   1:  PR[91,1] = PR[90,1] + 0.629;
   1:L PR[91] R[100]mm/sec CNT100;
   1:  PR[91,1] = PR[90,1] + 1.561;
   1:  PR[91,2] = PR[90,2] + -23.325;
   1:L PR[91] R[100]mm/sec CNT100;
   1:  PR[91,1] = PR[90,1] + 7.477;
   1:  PR[91,2] = PR[90,2] + -23.910;
   1:L PR[91] R[100]mm/sec CNT100;
   1:  PR[91,1] = PR[90,1] + 8.164;
   1:  PR[91,2] = PR[90,2] + -23.821;
   1:L PR[91] R[100]mm/sec CNT100;
   1:  PR[91,1] = PR[90,1] + 13.666;
   1:  PR[91,2] = PR[90,2] + -22.946;
   1:L PR[91] R[100]mm/sec CNT100;
   1:  PR[91,1] = PR[90,1] + 14.550;
   1:  PR[91,2] = PR[90,2] + -22.590;
   1:L PR[91] R[100]mm/sec CNT100;
   1:  PR[91,1] = PR[90,1] + 19.392;
   1:  PR[91,2] = PR[90,2] + -20.484;
   1:L PR[91] R[100]mm/sec CNT100;
   1:  PR[91,1] = PR[90,1] + 20.346;
   1:  PR[91,2] = PR[90,2] + -19.776;
   1:L PR[91] R[100]mm/sec CNT100;
   1:  PR[91,1] = PR[90,1] + 24.273;
   1:  PR[91,2] = PR[90,2] + -16.705;
   1:L PR[91] R[100]mm/sec CNT100;
   1:  PR[91,1] = PR[90,1] + 25.132;
   1:  PR[91,2] = PR[90,2] + -15.619;
   1:L PR[91] R[100]mm/sec CNT100;
   1:  PR[91,1] = PR[90,1] + 28.000;
   1:  PR[91,2] = PR[90,2] + -11.846;
   1:L PR[91] R[100]mm/sec CNT100;
   1:  PR[91,1] = PR[90,1] + 28.598;
   1:  PR[91,2] = PR[90,2] + -10.471;
   1:L PR[91] R[100]mm/sec CNT100;
   1:  PR[91,1] = PR[90,1] + 30.330;
   1:  PR[91,2] = PR[90,2] + -6.297;
   1:L PR[91] R[100]mm/sec CNT100;
   1:  PR[91,1] = PR[90,1] + 30.542;
   1:  PR[91,2] = PR[90,2] + -4.725;
   1:L PR[91] R[100]mm/sec CNT100;
   1:  PR[91,1] = PR[90,1] + 30.756;
   1:  PR[91,2] = PR[90,2] + -2.568;
   1:L PR[91] R[100]mm/sec CNT100;
   1:  PR[91,1] = PR[90,1] + 31.056;
   1:  PR[91,2] = PR[90,2] + -0.286;
   1:L PR[91] R[100]mm/sec CNT100;
   1:  PR[91,1] = PR[90,1] + 30.904;
   1:  PR[91,2] = PR[90,2] + 1.310;
   1:L PR[91] R[100]mm/sec CNT100;
   1:  PR[91,1] = PR[90,1] + 30.330;
   1:  PR[91,2] = PR[90,2] + 5.670;
   1:L PR[91] R[100]mm/sec CNT100;
   1:  PR[91,1] = PR[90,1] + 28.603;
   1:  PR[91,2] = PR[90,2] + 9.838;
   1:L PR[91] R[100]mm/sec CNT100;
   1:  PR[91,1] = PR[90,1] + 28.006;
   1:  PR[91,2] = PR[90,2] + 11.211;
   1:L PR[91] R[100]mm/sec CNT100;
   1:  PR[91,1] = PR[90,1] + 25.143;
   1:  PR[91,2] = PR[90,2] + 14.983;
   1:L PR[91] R[100]mm/sec CNT100;
   1:  PR[91,1] = PR[90,1] + 24.286;
   1:  PR[91,2] = PR[90,2] + 16.068;
   1:L PR[91] R[100]mm/sec CNT100;
   1:  PR[91,1] = PR[90,1] + 20.366;
   1:  PR[91,2] = PR[90,2] + 19.139;
   1:L PR[91] R[100]mm/sec CNT100;
   1:  PR[91,1] = PR[90,1] + 19.413;
   1:  PR[91,2] = PR[90,2] + 19.847;
   1:L PR[91] R[100]mm/sec CNT100;
   1:  PR[91,1] = PR[90,1] + 14.579;
   1:  PR[91,2] = PR[90,2] + 21.956;
   1:L PR[91] R[100]mm/sec CNT100;
   1:  PR[91,1] = PR[90,1] + 13.695;
   1:  PR[91,2] = PR[90,2] + 22.313;
   1:L PR[91] R[100]mm/sec CNT100;
   1:  PR[91,1] = PR[90,1] + 8.201;
   1:  PR[91,2] = PR[90,2] + 23.194;
   1:L PR[91] R[100]mm/sec CNT100;
   1:  PR[91,1] = PR[90,1] + 7.513;
   1:  PR[91,2] = PR[90,2] + 23.285;
   1:L PR[91] R[100]mm/sec CNT100;
   1:  PR[91,1] = PR[90,1] + 1.597;
   1:  PR[91,2] = PR[90,2] + 22.714;
   1:L PR[91] R[100]mm/sec CNT100;
   1:  PR[91,1] = PR[90,1] + 1.222;
   1:  PR[91,2] = PR[90,2] + 22.667;
   1:L PR[91] R[100]mm/sec CNT100;
   1:  PR[91,1] = PR[90,1] + 0.703;
   1:  PR[91,2] = PR[90,2] + 22.501;
   1:L PR[91] R[100]mm/sec CNT100;
   1:  PR[91] = PR[90];
   1:  PR[91,1] = PR[90,1] + -0.529;
   1:  PR[91,2] = PR[90,2] + 22.670;
   1:  PR[91,3] = PR[90,3] + 57.035;
   1:L PR[91] R[100]mm/sec CNT100;
   1:  PR[91,1] = PR[90,1] + -0.847;
   1:  PR[91,2] = PR[90,2] + 22.772;
   1:L PR[91] R[100]mm/sec CNT100;
   1:  PR[91,1] = PR[90,1] + -0.976;
   1:  PR[91,2] = PR[90,2] + 22.788;
   1:L PR[91] R[100]mm/sec CNT100;
   1:  PR[91,1] = PR[90,1] + -7.156;
   1:  PR[91,2] = PR[90,2] + 23.384;
   1:L PR[91] R[100]mm/sec CNT100;
   1:  PR[91,1] = PR[90,1] + -7.594;
   1:  PR[91,2] = PR[90,2] + 23.327;
   1:L PR[91] R[100]mm/sec CNT100;
   1:  PR[91,1] = PR[90,1] + -13.353;
   1:  PR[91,2] = PR[90,2] + 22.404;
   1:L PR[91] R[100]mm/sec CNT100;
   1:  PR[91,1] = PR[90,1] + -13.996;
   1:  PR[91,2] = PR[90,2] + 22.143;
   1:L PR[91] R[100]mm/sec CNT100;
   1:  PR[91,1] = PR[90,1] + -19.083;
   1:  PR[91,2] = PR[90,2] + 19.924;
   1:L PR[91] R[100]mm/sec CNT100;
   1:  PR[91,1] = PR[90,1] + -19.826;
   1:  PR[91,2] = PR[90,2] + 19.372;
   1:L PR[91] R[100]mm/sec CNT100;
   1:  PR[91,1] = PR[90,1] + -23.967;
   1:  PR[91,2] = PR[90,2] + 16.128;
   1:L PR[91] R[100]mm/sec CNT100;
   1:  PR[91,1] = PR[90,1] + -24.660;
   1:  PR[91,2] = PR[90,2] + 15.252;
   1:L PR[91] R[100]mm/sec CNT100;
   1:  PR[91,1] = PR[90,1] + -27.694;
   1:  PR[91,2] = PR[90,2] + 11.258;
   1:L PR[91] R[100]mm/sec CNT100;
   1:  PR[91,1] = PR[90,1] + -28.187;
   1:  PR[91,2] = PR[90,2] + 10.118;
   1:L PR[91] R[100]mm/sec CNT100;
   1:  PR[91,1] = PR[90,1] + -30.024;
   1:  PR[91,2] = PR[90,2] + 5.680;
   1:L PR[91] R[100]mm/sec CNT100;
   1:  PR[91,1] = PR[90,1] + -30.201;
   1:  PR[91,2] = PR[90,2] + 4.374;
   1:L PR[91] R[100]mm/sec CNT100;
   1:  PR[91,1] = PR[90,1] + -30.383;
   1:  PR[91,2] = PR[90,2] + 2.537;
   1:L PR[91] R[100]mm/sec CNT100;
   1:  PR[91,1] = PR[90,1] + -30.761;
   1:  PR[91,2] = PR[90,2] + -0.338;
   1:L PR[91] R[100]mm/sec CNT100;
   1:  PR[91,1] = PR[90,1] + -30.632;
   1:  PR[91,2] = PR[90,2] + -1.679;
   1:L PR[91] R[100]mm/sec CNT100;
   1:  PR[91,1] = PR[90,1] + -30.021;
   1:  PR[91,2] = PR[90,2] + -6.312;
   1:L PR[91] R[100]mm/sec CNT100;
   1:  PR[91,1] = PR[90,1] + -28.182;
   1:  PR[91,2] = PR[90,2] + -10.752;
   1:L PR[91] R[100]mm/sec CNT100;
   1:  PR[91,1] = PR[90,1] + -27.688;
   1:  PR[91,2] = PR[90,2] + -11.893;
   1:L PR[91] R[100]mm/sec CNT100;
   1:  PR[91,1] = PR[90,1] + -24.649;
   1:  PR[91,2] = PR[90,2] + -15.889;
   1:L PR[91] R[100]mm/sec CNT100;
   1:  PR[91,1] = PR[90,1] + -23.954;
   1:  PR[91,2] = PR[90,2] + -16.765;
   1:L PR[91] R[100]mm/sec CNT100;
   1:  PR[91,1] = PR[90,1] + -19.805;
   1:  PR[91,2] = PR[90,2] + -20.009;
   1:L PR[91] R[100]mm/sec CNT100;
   1:  PR[91,1] = PR[90,1] + -19.062;
   1:  PR[91,2] = PR[90,2] + -20.560;
   1:L PR[91] R[100]mm/sec CNT100;
   1:  PR[91,1] = PR[90,1] + -13.967;
   1:  PR[91,2] = PR[90,2] + -22.777;
   1:L PR[91] R[100]mm/sec CNT100;
   1:  PR[91,1] = PR[90,1] + -13.323;
   1:  PR[91,2] = PR[90,2] + -23.036;
   1:L PR[91] R[100]mm/sec CNT100;
   1:  PR[91,1] = PR[90,1] + -7.557;
   1:  PR[91,2] = PR[90,2] + -23.953;
   1:L PR[91] R[100]mm/sec CNT100;
   1:  PR[91,1] = PR[90,1] + -7.120;
   1:  PR[91,2] = PR[90,2] + -24.009;
   1:L PR[91] R[100]mm/sec CNT100;
   1:  PR[91,1] = PR[90,1] + -0.879;
   1:  PR[91,2] = PR[90,2] + -23.392;
   1:L PR[91] R[100]mm/sec CNT100;
   1:  PR[91,1] = PR[90,1] + -0.799;
   1:  PR[91,2] = PR[90,2] + -23.382;
   1:L PR[91] R[100]mm/sec CNT100;
   1:  PR[91,1] = PR[90,1] + -0.525;
   1:  PR[91,2] = PR[90,2] + -23.296;
   1:L PR[91] R[100]mm/sec CNT100;
   1:  PR[91,1] = PR[90,1] + 0.614;
   1:L PR[91] R[100]mm/sec CNT100;
   1:  PR[91,1] = PR[90,1] + 1.097;
   1:  PR[91,2] = PR[90,2] + -23.398;
   1:L PR[91] R[100]mm/sec CNT100;
   1:  PR[91,1] = PR[90,1] + 7.278;
   1:  PR[91,2] = PR[90,2] + -24.009;
   1:L PR[91] R[100]mm/sec CNT100;
   1:  PR[91,1] = PR[90,1] + 7.716;
   1:  PR[91,2] = PR[90,2] + -23.953;
   1:L PR[91] R[100]mm/sec CNT100;
   1:  PR[91,1] = PR[90,1] + 13.481;
   1:  PR[91,2] = PR[90,2] + -23.036;
   1:L PR[91] R[100]mm/sec CNT100;
   1:  PR[91,1] = PR[90,1] + 14.126;
   1:  PR[91,2] = PR[90,2] + -22.776;
   1:L PR[91] R[100]mm/sec CNT100;
   1:  PR[91,1] = PR[90,1] + 19.220;
   1:  PR[91,2] = PR[90,2] + -20.561;
   1:L PR[91] R[100]mm/sec CNT100;
   1:  PR[91,1] = PR[90,1] + 19.963;
   1:  PR[91,2] = PR[90,2] + -20.009;
   1:L PR[91] R[100]mm/sec CNT100;
   1:  PR[91,1] = PR[90,1] + 24.111;
   1:  PR[91,2] = PR[90,2] + -16.765;
   1:L PR[91] R[100]mm/sec CNT100;
   1:  PR[91,1] = PR[90,1] + 24.806;
   1:  PR[91,2] = PR[90,2] + -15.887;
   1:L PR[91] R[100]mm/sec CNT100;
   1:  PR[91,1] = PR[90,1] + 27.845;
   1:  PR[91,2] = PR[90,2] + -11.889;
   1:L PR[91] R[100]mm/sec CNT100;
   1:  PR[91,1] = PR[90,1] + 28.340;
   1:  PR[91,2] = PR[90,2] + -10.752;
   1:L PR[91] R[100]mm/sec CNT100;
   1:  PR[91,1] = PR[90,1] + 30.179;
   1:  PR[91,2] = PR[90,2] + -6.318;
   1:L PR[91] R[100]mm/sec CNT100;
   1:  PR[91,1] = PR[90,1] + 30.357;
   1:  PR[91,2] = PR[90,2] + -5.007;
   1:L PR[91] R[100]mm/sec CNT100;
   1:  PR[91,1] = PR[90,1] + 30.539;
   1:  PR[91,2] = PR[90,2] + -3.166;
   1:L PR[91] R[100]mm/sec CNT100;
   1:  PR[91,1] = PR[90,1] + 30.918;
   1:  PR[91,2] = PR[90,2] + -0.286;
   1:L PR[91] R[100]mm/sec CNT100;
   1:  PR[91,1] = PR[90,1] + 30.790;
   1:  PR[91,2] = PR[90,2] + 1.057;
   1:L PR[91] R[100]mm/sec CNT100;
   1:  PR[91,1] = PR[90,1] + 30.180;
   1:  PR[91,2] = PR[90,2] + 5.690;
   1:L PR[91] R[100]mm/sec CNT100;
   1:  PR[91,1] = PR[90,1] + 28.344;
   1:  PR[91,2] = PR[90,2] + 10.118;
   1:L PR[91] R[100]mm/sec CNT100;
   1:  PR[91,1] = PR[90,1] + 27.851;
   1:  PR[91,2] = PR[90,2] + 11.254;
   1:L PR[91] R[100]mm/sec CNT100;
   1:  PR[91,1] = PR[90,1] + 24.817;
   1:  PR[91,2] = PR[90,2] + 15.251;
   1:L PR[91] R[100]mm/sec CNT100;
   1:  PR[91,1] = PR[90,1] + 24.123;
   1:  PR[91,2] = PR[90,2] + 16.128;
   1:L PR[91] R[100]mm/sec CNT100;
   1:  PR[91,1] = PR[90,1] + 19.983;
   1:  PR[91,2] = PR[90,2] + 19.372;
   1:L PR[91] R[100]mm/sec CNT100;
   1:  PR[91,1] = PR[90,1] + 19.241;
   1:  PR[91,2] = PR[90,2] + 19.924;
   1:L PR[91] R[100]mm/sec CNT100;
   1:  PR[91,1] = PR[90,1] + 14.154;
   1:  PR[91,2] = PR[90,2] + 22.143;
   1:L PR[91] R[100]mm/sec CNT100;
   1:  PR[91,1] = PR[90,1] + 13.511;
   1:  PR[91,2] = PR[90,2] + 22.403;
   1:L PR[91] R[100]mm/sec CNT100;
   1:  PR[91,1] = PR[90,1] + 7.752;
   1:  PR[91,2] = PR[90,2] + 23.327;
   1:L PR[91] R[100]mm/sec CNT100;
   1:  PR[91,1] = PR[90,1] + 7.314;
   1:  PR[91,2] = PR[90,2] + 23.384;
   1:L PR[91] R[100]mm/sec CNT100;
   1:  PR[91,1] = PR[90,1] + 1.135;
   1:  PR[91,2] = PR[90,2] + 22.788;
   1:L PR[91] R[100]mm/sec CNT100;
   1:  PR[91,1] = PR[90,1] + 1.006;
   1:  PR[91,2] = PR[90,2] + 22.772;
   1:L PR[91] R[100]mm/sec CNT100;
   1:  PR[91,1] = PR[90,1] + 0.688;
   1:  PR[91,2] = PR[90,2] + 22.670;
   1:L PR[91] R[100]mm/sec CNT100;
   1:  PR[91] = PR[90];
   1:  PR[91,1] = PR[90,1] + -0.359;
   1:  PR[91,2] = PR[90,2] + 22.840;
   1:  PR[91,3] = PR[90,3] + 57.645;
   1:L PR[91] R[100]mm/sec CNT100;
   1:  PR[91,1] = PR[90,1] + -6.957;
   1:  PR[91,2] = PR[90,2] + 23.484;
   1:L PR[91] R[100]mm/sec CNT100;
   1:  PR[91,1] = PR[90,1] + -7.145;
   1:  PR[91,2] = PR[90,2] + 23.459;
   1:L PR[91] R[100]mm/sec CNT100;
   1:  PR[91,1] = PR[90,1] + -13.168;
   1:  PR[91,2] = PR[90,2] + 22.494;
   1:L PR[91] R[100]mm/sec CNT100;
   1:  PR[91,1] = PR[90,1] + -13.572;
   1:  PR[91,2] = PR[90,2] + 22.330;
   1:L PR[91] R[100]mm/sec CNT100;
   1:  PR[91,1] = PR[90,1] + -18.911;
   1:  PR[91,2] = PR[90,2] + 20.001;
   1:L PR[91] R[100]mm/sec CNT100;
   1:  PR[91,1] = PR[90,1] + -19.443;
   1:  PR[91,2] = PR[90,2] + 19.605;
   1:L PR[91] R[100]mm/sec CNT100;
   1:  PR[91,1] = PR[90,1] + -23.805;
   1:  PR[91,2] = PR[90,2] + 16.189;
   1:L PR[91] R[100]mm/sec CNT100;
   1:  PR[91,1] = PR[90,1] + -24.335;
   1:  PR[91,2] = PR[90,2] + 15.519;
   1:L PR[91] R[100]mm/sec CNT100;
   1:  PR[91,1] = PR[90,1] + -27.539;
   1:  PR[91,2] = PR[90,2] + 11.301;
   1:L PR[91] R[100]mm/sec CNT100;
   1:  PR[91,1] = PR[90,1] + -27.929;
   1:  PR[91,2] = PR[90,2] + 10.399;
   1:L PR[91] R[100]mm/sec CNT100;
   1:  PR[91,1] = PR[90,1] + -29.874;
   1:  PR[91,2] = PR[90,2] + 5.701;
   1:L PR[91] R[100]mm/sec CNT100;
   1:  PR[91,1] = PR[90,1] + -30.015;
   1:  PR[91,2] = PR[90,2] + 4.655;
   1:L PR[91] R[100]mm/sec CNT100;
   1:  PR[91,1] = PR[90,1] + -30.166;
   1:  PR[91,2] = PR[90,2] + 3.133;
   1:L PR[91] R[100]mm/sec CNT100;
   1:  PR[91,1] = PR[90,1] + -30.622;
   1:  PR[91,2] = PR[90,2] + -0.338;
   1:L PR[91] R[100]mm/sec CNT100;
   1:  PR[91,1] = PR[90,1] + -30.518;
   1:  PR[91,2] = PR[90,2] + -1.427;
   1:L PR[91] R[100]mm/sec CNT100;
   1:  PR[91,1] = PR[90,1] + -29.871;
   1:  PR[91,2] = PR[90,2] + -6.333;
   1:L PR[91] R[100]mm/sec CNT100;
   1:  PR[91,1] = PR[90,1] + -27.923;
   1:  PR[91,2] = PR[90,2] + -11.033;
   1:L PR[91] R[100]mm/sec CNT100;
   1:  PR[91,1] = PR[90,1] + -27.533;
   1:  PR[91,2] = PR[90,2] + -11.936;
   1:L PR[91] R[100]mm/sec CNT100;
   1:  PR[91,1] = PR[90,1] + -24.323;
   1:  PR[91,2] = PR[90,2] + -16.156;
   1:L PR[91] R[100]mm/sec CNT100;
   1:  PR[91,1] = PR[90,1] + -23.792;
   1:  PR[91,2] = PR[90,2] + -16.826;
   1:L PR[91] R[100]mm/sec CNT100;
   1:  PR[91,1] = PR[90,1] + -19.423;
   1:  PR[91,2] = PR[90,2] + -20.242;
   1:L PR[91] R[100]mm/sec CNT100;
   1:  PR[91,1] = PR[90,1] + -18.890;
   1:  PR[91,2] = PR[90,2] + -20.637;
   1:L PR[91] R[100]mm/sec CNT100;
   1:  PR[91,1] = PR[90,1] + -13.543;
   1:  PR[91,2] = PR[90,2] + -22.964;
   1:L PR[91] R[100]mm/sec CNT100;
   1:  PR[91,1] = PR[90,1] + -13.139;
   1:  PR[91,2] = PR[90,2] + -23.126;
   1:L PR[91] R[100]mm/sec CNT100;
   1:  PR[91,1] = PR[90,1] + -7.108;
   1:  PR[91,2] = PR[90,2] + -24.085;
   1:L PR[91] R[100]mm/sec CNT100;
   1:  PR[91,1] = PR[90,1] + -6.921;
   1:  PR[91,2] = PR[90,2] + -24.109;
   1:L PR[91] R[100]mm/sec CNT100;
   1:  PR[91,1] = PR[90,1] + -0.762;
   1:  PR[91,2] = PR[90,2] + -23.500;
   1:L PR[91] R[100]mm/sec CNT100;
   1:  PR[91,1] = PR[90,1] + -0.352;
   1:  PR[91,2] = PR[90,2] + -23.464;
   1:L PR[91] R[100]mm/sec CNT100;
   1:  PR[91,1] = PR[90,1] + 0.519;
   1:L PR[91] R[100]mm/sec CNT100;
   1:  PR[91,1] = PR[90,1] + 7.079;
   1:  PR[91,2] = PR[90,2] + -24.109;
   1:L PR[91] R[100]mm/sec CNT100;
   1:  PR[91,1] = PR[90,1] + 7.266;
   1:  PR[91,2] = PR[90,2] + -24.085;
   1:L PR[91] R[100]mm/sec CNT100;
   1:  PR[91,1] = PR[90,1] + 13.297;
   1:  PR[91,2] = PR[90,2] + -23.125;
   1:L PR[91] R[100]mm/sec CNT100;
   1:  PR[91,1] = PR[90,1] + 13.701;
   1:  PR[91,2] = PR[90,2] + -22.963;
   1:L PR[91] R[100]mm/sec CNT100;
   1:  PR[91,1] = PR[90,1] + 19.048;
   1:  PR[91,2] = PR[90,2] + -20.638;
   1:L PR[91] R[100]mm/sec CNT100;
   1:  PR[91,1] = PR[90,1] + 19.581;
   1:  PR[91,2] = PR[90,2] + -20.242;
   1:L PR[91] R[100]mm/sec CNT100;
   1:  PR[91,1] = PR[90,1] + 23.948;
   1:  PR[91,2] = PR[90,2] + -16.826;
   1:L PR[91] R[100]mm/sec CNT100;
   1:  PR[91,1] = PR[90,1] + 24.480;
   1:  PR[91,2] = PR[90,2] + -16.155;
   1:L PR[91] R[100]mm/sec CNT100;
   1:  PR[91,1] = PR[90,1] + 27.690;
   1:  PR[91,2] = PR[90,2] + -11.931;
   1:L PR[91] R[100]mm/sec CNT100;
   1:  PR[91,1] = PR[90,1] + 28.081;
   1:  PR[91,2] = PR[90,2] + -11.033;
   1:L PR[91] R[100]mm/sec CNT100;
   1:  PR[91,1] = PR[90,1] + 30.029;
   1:  PR[91,2] = PR[90,2] + -6.338;
   1:L PR[91] R[100]mm/sec CNT100;
   1:  PR[91,1] = PR[90,1] + 30.171;
   1:  PR[91,2] = PR[90,2] + -5.288;
   1:L PR[91] R[100]mm/sec CNT100;
   1:  PR[91,1] = PR[90,1] + 30.322;
   1:  PR[91,2] = PR[90,2] + -3.763;
   1:L PR[91] R[100]mm/sec CNT100;
   1:  PR[91,1] = PR[90,1] + 30.779;
   1:  PR[91,2] = PR[90,2] + -0.286;
   1:L PR[91] R[100]mm/sec CNT100;
   1:  PR[91,1] = PR[90,1] + 30.675;
   1:  PR[91,2] = PR[90,2] + 0.805;
   1:L PR[91] R[100]mm/sec CNT100;
   1:  PR[91,1] = PR[90,1] + 30.029;
   1:  PR[91,2] = PR[90,2] + 5.711;
   1:L PR[91] R[100]mm/sec CNT100;
   1:  PR[91,1] = PR[90,1] + 28.086;
   1:  PR[91,2] = PR[90,2] + 10.399;
   1:L PR[91] R[100]mm/sec CNT100;
   1:  PR[91,1] = PR[90,1] + 27.696;
   1:  PR[91,2] = PR[90,2] + 11.297;
   1:L PR[91] R[100]mm/sec CNT100;
   1:  PR[91,1] = PR[90,1] + 24.491;
   1:  PR[91,2] = PR[90,2] + 15.518;
   1:L PR[91] R[100]mm/sec CNT100;
   1:  PR[91,1] = PR[90,1] + 23.961;
   1:  PR[91,2] = PR[90,2] + 16.189;
   1:L PR[91] R[100]mm/sec CNT100;
   1:  PR[91,1] = PR[90,1] + 19.601;
   1:  PR[91,2] = PR[90,2] + 19.606;
   1:L PR[91] R[100]mm/sec CNT100;
   1:  PR[91,1] = PR[90,1] + 19.069;
   1:  PR[91,2] = PR[90,2] + 20.001;
   1:L PR[91] R[100]mm/sec CNT100;
   1:  PR[91,1] = PR[90,1] + 13.731;
   1:  PR[91,2] = PR[90,2] + 22.330;
   1:L PR[91] R[100]mm/sec CNT100;
   1:  PR[91,1] = PR[90,1] + 13.326;
   1:  PR[91,2] = PR[90,2] + 22.493;
   1:L PR[91] R[100]mm/sec CNT100;
   1:  PR[91,1] = PR[90,1] + 7.303;
   1:  PR[91,2] = PR[90,2] + 23.459;
   1:L PR[91] R[100]mm/sec CNT100;
   1:  PR[91,1] = PR[90,1] + 7.115;
   1:  PR[91,2] = PR[90,2] + 23.484;
   1:L PR[91] R[100]mm/sec CNT100;
   1:  PR[91,1] = PR[90,1] + 0.518;
   1:  PR[91,2] = PR[90,2] + 22.840;
   1:L PR[91] R[100]mm/sec CNT100;
   1:  PR[91] = PR[90];
   1:  PR[91,1] = PR[90,1] + -0.337;
   1:  PR[91,2] = PR[90,2] + 23.004;
   1:  PR[91,3] = PR[90,3] + 58.255;
   1:L PR[91] R[100]mm/sec CNT100;
   1:  PR[91,1] = PR[90,1] + -4.502;
   1:  PR[91,2] = PR[90,2] + 23.366;
   1:L PR[91] R[100]mm/sec CNT100;
   1:  PR[91,1] = PR[90,1] + -6.737;
   1:  PR[91,2] = PR[90,2] + 23.581;
   1:L PR[91] R[100]mm/sec CNT100;
   1:  PR[91,1] = PR[90,1] + -12.984;
   1:  PR[91,2] = PR[90,2] + 22.584;
   1:L PR[91] R[100]mm/sec CNT100;
   1:  PR[91,1] = PR[90,1] + -13.148;
   1:  PR[91,2] = PR[90,2] + 22.517;
   1:L PR[91] R[100]mm/sec CNT100;
   1:  PR[91,1] = PR[90,1] + -18.739;
   1:  PR[91,2] = PR[90,2] + 20.078;
   1:L PR[91] R[100]mm/sec CNT100;
   1:  PR[91,1] = PR[90,1] + -19.061;
   1:  PR[91,2] = PR[90,2] + 19.839;
   1:L PR[91] R[100]mm/sec CNT100;
   1:  PR[91,1] = PR[90,1] + -23.642;
   1:  PR[91,2] = PR[90,2] + 16.250;
   1:L PR[91] R[100]mm/sec CNT100;
   1:  PR[91,1] = PR[90,1] + -24.009;
   1:  PR[91,2] = PR[90,2] + 15.787;
   1:L PR[91] R[100]mm/sec CNT100;
   1:  PR[91,1] = PR[90,1] + -27.384;
   1:  PR[91,2] = PR[90,2] + 11.344;
   1:L PR[91] R[100]mm/sec CNT100;
   1:  PR[91,1] = PR[90,1] + -27.671;
   1:  PR[91,2] = PR[90,2] + 10.681;
   1:L PR[91] R[100]mm/sec CNT100;
   1:  PR[91,1] = PR[90,1] + -29.723;
   1:  PR[91,2] = PR[90,2] + 5.722;
   1:L PR[91] R[100]mm/sec CNT100;
   1:  PR[91,1] = PR[90,1] + -29.830;
   1:  PR[91,2] = PR[90,2] + 4.936;
   1:L PR[91] R[100]mm/sec CNT100;
   1:  PR[91,1] = PR[90,1] + -29.949;
   1:  PR[91,2] = PR[90,2] + 3.729;
   1:L PR[91] R[100]mm/sec CNT100;
   1:  PR[91,1] = PR[90,1] + -30.483;
   1:  PR[91,2] = PR[90,2] + -0.338;
   1:L PR[91] R[100]mm/sec CNT100;
   1:  PR[91,1] = PR[90,1] + -30.403;
   1:  PR[91,2] = PR[90,2] + -1.175;
   1:L PR[91] R[100]mm/sec CNT100;
   1:  PR[91,1] = PR[90,1] + -29.720;
   1:  PR[91,2] = PR[90,2] + -6.354;
   1:L PR[91] R[100]mm/sec CNT100;
   1:  PR[91,1] = PR[90,1] + -27.665;
   1:  PR[91,2] = PR[90,2] + -11.315;
   1:L PR[91] R[100]mm/sec CNT100;
   1:  PR[91,1] = PR[90,1] + -27.378;
   1:  PR[91,2] = PR[90,2] + -11.978;
   1:L PR[91] R[100]mm/sec CNT100;
   1:  PR[91,1] = PR[90,1] + -23.997;
   1:  PR[91,2] = PR[90,2] + -16.424;
   1:L PR[91] R[100]mm/sec CNT100;
   1:  PR[91,1] = PR[90,1] + -23.630;
   1:  PR[91,2] = PR[90,2] + -16.886;
   1:L PR[91] R[100]mm/sec CNT100;
   1:  PR[91,1] = PR[90,1] + -19.040;
   1:  PR[91,2] = PR[90,2] + -20.476;
   1:L PR[91] R[100]mm/sec CNT100;
   1:  PR[91,1] = PR[90,1] + -18.719;
   1:  PR[91,2] = PR[90,2] + -20.714;
   1:L PR[91] R[100]mm/sec CNT100;
   1:  PR[91,1] = PR[90,1] + -12.936;
   1:  PR[91,2] = PR[90,2] + -23.219;
   1:L PR[91] R[100]mm/sec CNT100;
   1:  PR[91,1] = PR[90,1] + -6.715;
   1:  PR[91,2] = PR[90,2] + -24.208;
   1:L PR[91] R[100]mm/sec CNT100;
   1:  PR[91,1] = PR[90,1] + -4.834;
   1:  PR[91,2] = PR[90,2] + -24.022;
   1:L PR[91] R[100]mm/sec CNT100;
   1:  PR[91,1] = PR[90,1] + -0.338;
   1:  PR[91,2] = PR[90,2] + -23.626;
   1:L PR[91] R[100]mm/sec CNT100;
   1:  PR[91,1] = PR[90,1] + 0.497;
   1:L PR[91] R[100]mm/sec CNT100;
   1:  PR[91,1] = PR[90,1] + 4.986;
   1:  PR[91,2] = PR[90,2] + -24.021;
   1:L PR[91] R[100]mm/sec CNT100;
   1:  PR[91,1] = PR[90,1] + 6.860;
   1:  PR[91,2] = PR[90,2] + -24.206;
   1:L PR[91] R[100]mm/sec CNT100;
   1:  PR[91,1] = PR[90,1] + 13.114;
   1:  PR[91,2] = PR[90,2] + -23.215;
   1:L PR[91] R[100]mm/sec CNT100;
   1:  PR[91,1] = PR[90,1] + 13.277;
   1:  PR[91,2] = PR[90,2] + -23.149;
   1:L PR[91] R[100]mm/sec CNT100;
   1:  PR[91,1] = PR[90,1] + 18.876;
   1:  PR[91,2] = PR[90,2] + -20.714;
   1:L PR[91] R[100]mm/sec CNT100;
   1:  PR[91,1] = PR[90,1] + 19.198;
   1:  PR[91,2] = PR[90,2] + -20.476;
   1:L PR[91] R[100]mm/sec CNT100;
   1:  PR[91,1] = PR[90,1] + 23.786;
   1:  PR[91,2] = PR[90,2] + -16.886;
   1:L PR[91] R[100]mm/sec CNT100;
   1:  PR[91,1] = PR[90,1] + 24.154;
   1:  PR[91,2] = PR[90,2] + -16.423;
   1:L PR[91] R[100]mm/sec CNT100;
   1:  PR[91,1] = PR[90,1] + 27.535;
   1:  PR[91,2] = PR[90,2] + -11.974;
   1:L PR[91] R[100]mm/sec CNT100;
   1:  PR[91,1] = PR[90,1] + 27.823;
   1:  PR[91,2] = PR[90,2] + -11.313;
   1:L PR[91] R[100]mm/sec CNT100;
   1:  PR[91,1] = PR[90,1] + 29.878;
   1:  PR[91,2] = PR[90,2] + -6.359;
   1:L PR[91] R[100]mm/sec CNT100;
   1:  PR[91,1] = PR[90,1] + 29.985;
   1:  PR[91,2] = PR[90,2] + -5.569;
   1:L PR[91] R[100]mm/sec CNT100;
   1:  PR[91,1] = PR[90,1] + 30.105;
   1:  PR[91,2] = PR[90,2] + -4.360;
   1:L PR[91] R[100]mm/sec CNT100;
   1:  PR[91,1] = PR[90,1] + 30.640;
   1:  PR[91,2] = PR[90,2] + -0.286;
   1:L PR[91] R[100]mm/sec CNT100;
   1:  PR[91,1] = PR[90,1] + 30.560;
   1:  PR[91,2] = PR[90,2] + 0.553;
   1:L PR[91] R[100]mm/sec CNT100;
   1:  PR[91,1] = PR[90,1] + 29.879;
   1:  PR[91,2] = PR[90,2] + 5.731;
   1:L PR[91] R[100]mm/sec CNT100;
   1:  PR[91,1] = PR[90,1] + 27.828;
   1:  PR[91,2] = PR[90,2] + 10.679;
   1:L PR[91] R[100]mm/sec CNT100;
   1:  PR[91,1] = PR[90,1] + 27.541;
   1:  PR[91,2] = PR[90,2] + 11.339;
   1:L PR[91] R[100]mm/sec CNT100;
   1:  PR[91,1] = PR[90,1] + 24.166;
   1:  PR[91,2] = PR[90,2] + 15.786;
   1:L PR[91] R[100]mm/sec CNT100;
   1:  PR[91,1] = PR[90,1] + 23.799;
   1:  PR[91,2] = PR[90,2] + 16.250;
   1:L PR[91] R[100]mm/sec CNT100;
   1:  PR[91,1] = PR[90,1] + 19.219;
   1:  PR[91,2] = PR[90,2] + 19.839;
   1:L PR[91] R[100]mm/sec CNT100;
   1:  PR[91,1] = PR[90,1] + 18.897;
   1:  PR[91,2] = PR[90,2] + 20.078;
   1:L PR[91] R[100]mm/sec CNT100;
   1:  PR[91,1] = PR[90,1] + 13.123;
   1:  PR[91,2] = PR[90,2] + 22.586;
   1:L PR[91] R[100]mm/sec CNT100;
   1:  PR[91,1] = PR[90,1] + 6.909;
   1:  PR[91,2] = PR[90,2] + 23.583;
   1:L PR[91] R[100]mm/sec CNT100;
   1:  PR[91,1] = PR[90,1] + 4.657;
   1:  PR[91,2] = PR[90,2] + 23.365;
   1:L PR[91] R[100]mm/sec CNT100;
   1:  PR[91,1] = PR[90,1] + 0.496;
   1:  PR[91,2] = PR[90,2] + 23.004;
   1:L PR[91] R[100]mm/sec CNT100;
   1:  PR[91] = PR[90];
   1:  PR[91,1] = PR[90,1] + -0.323;
   1:  PR[91,2] = PR[90,2] + 23.167;
   1:  PR[91,3] = PR[90,3] + 58.865;
   1:L PR[91] R[100]mm/sec CNT100;
   1:  PR[91,1] = PR[90,1] + -6.498;
   1:  PR[91,2] = PR[90,2] + 23.701;
   1:L PR[91] R[100]mm/sec CNT100;
   1:  PR[91,1] = PR[90,1] + -12.789;
   1:  PR[91,2] = PR[90,2] + 22.676;
   1:L PR[91] R[100]mm/sec CNT100;
   1:  PR[91,1] = PR[90,1] + -18.550;
   1:  PR[91,2] = PR[90,2] + 20.162;
   1:L PR[91] R[100]mm/sec CNT100;
   1:  PR[91,1] = PR[90,1] + -23.470;
   1:  PR[91,2] = PR[90,2] + 16.318;
   1:L PR[91] R[100]mm/sec CNT100;
   1:  PR[91,1] = PR[90,1] + -27.223;
   1:  PR[91,2] = PR[90,2] + 11.393;
   1:L PR[91] R[100]mm/sec CNT100;
   1:  PR[91,1] = PR[90,1] + -29.573;
   1:  PR[91,2] = PR[90,2] + 5.742;
   1:L PR[91] R[100]mm/sec CNT100;
   1:  PR[91,1] = PR[90,1] + -29.644;
   1:  PR[91,2] = PR[90,2] + 5.217;
   1:L PR[91] R[100]mm/sec CNT100;
   1:  PR[91,1] = PR[90,1] + -29.732;
   1:  PR[91,2] = PR[90,2] + 4.326;
   1:L PR[91] R[100]mm/sec CNT100;
   1:  PR[91,1] = PR[90,1] + -30.345;
   1:  PR[91,2] = PR[90,2] + -0.338;
   1:L PR[91] R[100]mm/sec CNT100;
   1:  PR[91,1] = PR[90,1] + -30.289;
   1:  PR[91,2] = PR[90,2] + -0.923;
   1:L PR[91] R[100]mm/sec CNT100;
   1:  PR[91,1] = PR[90,1] + -29.570;
   1:  PR[91,2] = PR[90,2] + -6.374;
   1:L PR[91] R[100]mm/sec CNT100;
   1:  PR[91,1] = PR[90,1] + -27.217;
   1:  PR[91,2] = PR[90,2] + -12.029;
   1:L PR[91] R[100]mm/sec CNT100;
   1:  PR[91,1] = PR[90,1] + -23.670;
   1:  PR[91,2] = PR[90,2] + -16.691;
   1:L PR[91] R[100]mm/sec CNT100;
   1:  PR[91,1] = PR[90,1] + -23.468;
   1:  PR[91,2] = PR[90,2] + -16.946;
   1:L PR[91] R[100]mm/sec CNT100;
   1:  PR[91,1] = PR[90,1] + -18.530;
   1:  PR[91,2] = PR[90,2] + -20.798;
   1:L PR[91] R[100]mm/sec CNT100;
   1:  PR[91,1] = PR[90,1] + -12.751;
   1:  PR[91,2] = PR[90,2] + -23.309;
   1:L PR[91] R[100]mm/sec CNT100;
   1:  PR[91,1] = PR[90,1] + -10.118;
   1:  PR[91,2] = PR[90,2] + -23.728;
   1:L PR[91] R[100]mm/sec CNT100;
   1:  PR[91,1] = PR[90,1] + -6.477;
   1:  PR[91,2] = PR[90,2] + -24.330;
   1:L PR[91] R[100]mm/sec CNT100;
   1:  PR[91,1] = PR[90,1] + -6.453;
   1:  PR[91,2] = PR[90,2] + -24.328;
   1:L PR[91] R[100]mm/sec CNT100;
   1:  PR[91,1] = PR[90,1] + -0.324;
   1:  PR[91,2] = PR[90,2] + -23.789;
   1:L PR[91] R[100]mm/sec CNT100;
   1:  PR[91,1] = PR[90,1] + 0.483;
   1:L PR[91] R[100]mm/sec CNT100;
   1:  PR[91,1] = PR[90,1] + 6.583;
   1:  PR[91,2] = PR[90,2] + -24.325;
   1:L PR[91] R[100]mm/sec CNT100;
   1:  PR[91,1] = PR[90,1] + 6.654;
   1:  PR[91,2] = PR[90,2] + -24.328;
   1:L PR[91] R[100]mm/sec CNT100;
   1:  PR[91,1] = PR[90,1] + 10.266;
   1:  PR[91,2] = PR[90,2] + -23.729;
   1:L PR[91] R[100]mm/sec CNT100;
   1:  PR[91,1] = PR[90,1] + 12.910;
   1:  PR[91,2] = PR[90,2] + -23.308;
   1:L PR[91] R[100]mm/sec CNT100;
   1:  PR[91,1] = PR[90,1] + 18.688;
   1:  PR[91,2] = PR[90,2] + -20.798;
   1:L PR[91] R[100]mm/sec CNT100;
   1:  PR[91,1] = PR[90,1] + 23.615;
   1:  PR[91,2] = PR[90,2] + -16.954;
   1:L PR[91] R[100]mm/sec CNT100;
   1:  PR[91,1] = PR[90,1] + 27.374;
   1:  PR[91,2] = PR[90,2] + -12.024;
   1:L PR[91] R[100]mm/sec CNT100;
   1:  PR[91,1] = PR[90,1] + 29.728;
   1:  PR[91,2] = PR[90,2] + -6.378;
   1:L PR[91] R[100]mm/sec CNT100;
   1:  PR[91,1] = PR[90,1] + 29.799;
   1:  PR[91,2] = PR[90,2] + -5.851;
   1:L PR[91] R[100]mm/sec CNT100;
   1:  PR[91,1] = PR[90,1] + 29.888;
   1:  PR[91,2] = PR[90,2] + -4.958;
   1:L PR[91] R[100]mm/sec CNT100;
   1:  PR[91,1] = PR[90,1] + 30.502;
   1:  PR[91,2] = PR[90,2] + -0.286;
   1:L PR[91] R[100]mm/sec CNT100;
   1:  PR[91,1] = PR[90,1] + 30.446;
   1:  PR[91,2] = PR[90,2] + 0.301;
   1:L PR[91] R[100]mm/sec CNT100;
   1:  PR[91,1] = PR[90,1] + 29.728;
   1:  PR[91,2] = PR[90,2] + 5.751;
   1:L PR[91] R[100]mm/sec CNT100;
   1:  PR[91,1] = PR[90,1] + 27.380;
   1:  PR[91,2] = PR[90,2] + 11.390;
   1:L PR[91] R[100]mm/sec CNT100;
   1:  PR[91,1] = PR[90,1] + 23.627;
   1:  PR[91,2] = PR[90,2] + 16.318;
   1:L PR[91] R[100]mm/sec CNT100;
   1:  PR[91,1] = PR[90,1] + 18.708;
   1:  PR[91,2] = PR[90,2] + 20.162;
   1:L PR[91] R[100]mm/sec CNT100;
   1:  PR[91,1] = PR[90,1] + 12.938;
   1:  PR[91,2] = PR[90,2] + 22.676;
   1:L PR[91] R[100]mm/sec CNT100;
   1:  PR[91,1] = PR[90,1] + 10.264;
   1:  PR[91,2] = PR[90,2] + 23.105;
   1:L PR[91] R[100]mm/sec CNT100;
   1:  PR[91,1] = PR[90,1] + 6.673;
   1:  PR[91,2] = PR[90,2] + 23.704;
   1:L PR[91] R[100]mm/sec CNT100;
   1:  PR[91,1] = PR[90,1] + 6.540;
   1:  PR[91,2] = PR[90,2] + 23.694;
   1:L PR[91] R[100]mm/sec CNT100;
   1:  PR[91,1] = PR[90,1] + 0.482;
   1:  PR[91,2] = PR[90,2] + 23.167;
   1:L PR[91] R[100]mm/sec CNT100;
   1:  PR[91] = PR[90];
   1:  PR[91,1] = PR[90,1] + -0.308;
   1:  PR[91,2] = PR[90,2] + 23.330;
   1:  PR[91,3] = PR[90,3] + 59.475;
   1:L PR[91] R[100]mm/sec CNT100;
   1:  PR[91,1] = PR[90,1] + -6.267;
   1:  PR[91,2] = PR[90,2] + 23.841;
   1:L PR[91] R[100]mm/sec CNT100;
   1:  PR[91,1] = PR[90,1] + -6.497;
   1:  PR[91,2] = PR[90,2] + 23.813;
   1:L PR[91] R[100]mm/sec CNT100;
   1:  PR[91,1] = PR[90,1] + -12.584;
   1:  PR[91,2] = PR[90,2] + 22.798;
   1:L PR[91] R[100]mm/sec CNT100;
   1:  PR[91,1] = PR[90,1] + -18.375;
   1:  PR[91,2] = PR[90,2] + 20.241;
   1:L PR[91] R[100]mm/sec CNT100;
   1:  PR[91,1] = PR[90,1] + -23.307;
   1:  PR[91,2] = PR[90,2] + 16.380;
   1:L PR[91] R[100]mm/sec CNT100;
   1:  PR[91,1] = PR[90,1] + -27.068;
   1:  PR[91,2] = PR[90,2] + 11.437;
   1:L PR[91] R[100]mm/sec CNT100;
   1:  PR[91,1] = PR[90,1] + -29.417;
   1:  PR[91,2] = PR[90,2] + 5.777;
   1:L PR[91] R[100]mm/sec CNT100;
   1:  PR[91,1] = PR[90,1] + -29.517;
   1:  PR[91,2] = PR[90,2] + 4.910;
   1:L PR[91] R[100]mm/sec CNT100;
   1:  PR[91,1] = PR[90,1] + -30.206;
   1:  PR[91,2] = PR[90,2] + -0.338;
   1:L PR[91] R[100]mm/sec CNT100;
   1:  PR[91,1] = PR[90,1] + -30.174;
   1:  PR[91,2] = PR[90,2] + -0.671;
   1:L PR[91] R[100]mm/sec CNT100;
   1:  PR[91,1] = PR[90,1] + -29.420;
   1:  PR[91,2] = PR[90,2] + -6.396;
   1:L PR[91] R[100]mm/sec CNT100;
   1:  PR[91,1] = PR[90,1] + -27.062;
   1:  PR[91,2] = PR[90,2] + -12.071;
   1:L PR[91] R[100]mm/sec CNT100;
   1:  PR[91,1] = PR[90,1] + -23.345;
   1:  PR[91,2] = PR[90,2] + -16.958;
   1:L PR[91] R[100]mm/sec CNT100;
   1:  PR[91,1] = PR[90,1] + -23.305;
   1:  PR[91,2] = PR[90,2] + -17.008;
   1:L PR[91] R[100]mm/sec CNT100;
   1:  PR[91,1] = PR[90,1] + -18.355;
   1:  PR[91,2] = PR[90,2] + -20.877;
   1:L PR[91] R[100]mm/sec CNT100;
   1:  PR[91,1] = PR[90,1] + -12.520;
   1:  PR[91,2] = PR[90,2] + -23.437;
   1:L PR[91] R[100]mm/sec CNT100;
   1:  PR[91,1] = PR[90,1] + -6.461;
   1:  PR[91,2] = PR[90,2] + -24.439;
   1:L PR[91] R[100]mm/sec CNT100;
   1:  PR[91,1] = PR[90,1] + -6.228;
   1:  PR[91,2] = PR[90,2] + -24.466;
   1:L PR[91] R[100]mm/sec CNT100;
   1:  PR[91,1] = PR[90,1] + -0.309;
   1:  PR[91,2] = PR[90,2] + -23.951;
   1:L PR[91] R[100]mm/sec CNT100;
   1:  PR[91,1] = PR[90,1] + 0.468;
   1:L PR[91] R[100]mm/sec CNT100;
   1:  PR[91,1] = PR[90,1] + 6.009;
   1:  PR[91,2] = PR[90,2] + -24.438;
   1:L PR[91] R[100]mm/sec CNT100;
   1:  PR[91,1] = PR[90,1] + 6.422;
   1:  PR[91,2] = PR[90,2] + -24.471;
   1:L PR[91] R[100]mm/sec CNT100;
   1:  PR[91,1] = PR[90,1] + 6.467;
   1:  PR[91,2] = PR[90,2] + -24.468;
   1:L PR[91] R[100]mm/sec CNT100;
   1:  PR[91,1] = PR[90,1] + 12.685;
   1:  PR[91,2] = PR[90,2] + -23.435;
   1:L PR[91] R[100]mm/sec CNT100;
   1:  PR[91,1] = PR[90,1] + 18.513;
   1:  PR[91,2] = PR[90,2] + -20.877;
   1:L PR[91] R[100]mm/sec CNT100;
   1:  PR[91,1] = PR[90,1] + 23.452;
   1:  PR[91,2] = PR[90,2] + -17.016;
   1:L PR[91] R[100]mm/sec CNT100;
   1:  PR[91,1] = PR[90,1] + 27.219;
   1:  PR[91,2] = PR[90,2] + -12.068;
   1:L PR[91] R[100]mm/sec CNT100;
   1:  PR[91,1] = PR[90,1] + 29.572;
   1:  PR[91,2] = PR[90,2] + -6.412;
   1:L PR[91] R[100]mm/sec CNT100;
   1:  PR[91,1] = PR[90,1] + 29.672;
   1:  PR[91,2] = PR[90,2] + -5.544;
   1:L PR[91] R[100]mm/sec CNT100;
   1:  PR[91,1] = PR[90,1] + 30.363;
   1:  PR[91,2] = PR[90,2] + -0.286;
   1:L PR[91] R[100]mm/sec CNT100;
   1:  PR[91,1] = PR[90,1] + 30.331;
   1:  PR[91,2] = PR[90,2] + 0.048;
   1:L PR[91] R[100]mm/sec CNT100;
   1:  PR[91,1] = PR[90,1] + 29.578;
   1:  PR[91,2] = PR[90,2] + 5.772;
   1:L PR[91] R[100]mm/sec CNT100;
   1:  PR[91,1] = PR[90,1] + 27.225;
   1:  PR[91,2] = PR[90,2] + 11.433;
   1:L PR[91] R[100]mm/sec CNT100;
   1:  PR[91,1] = PR[90,1] + 23.464;
   1:  PR[91,2] = PR[90,2] + 16.379;
   1:L PR[91] R[100]mm/sec CNT100;
   1:  PR[91,1] = PR[90,1] + 18.533;
   1:  PR[91,2] = PR[90,2] + 20.241;
   1:L PR[91] R[100]mm/sec CNT100;
   1:  PR[91,1] = PR[90,1] + 12.712;
   1:  PR[91,2] = PR[90,2] + 22.803;
   1:L PR[91] R[100]mm/sec CNT100;
   1:  PR[91,1] = PR[90,1] + 6.655;
   1:  PR[91,2] = PR[90,2] + 23.813;
   1:L PR[91] R[100]mm/sec CNT100;
   1:  PR[91,1] = PR[90,1] + 6.426;
   1:  PR[91,2] = PR[90,2] + 23.842;
   1:L PR[91] R[100]mm/sec CNT100;
   1:  PR[91,1] = PR[90,1] + 0.466;
   1:  PR[91,2] = PR[90,2] + 23.331;
   1:L PR[91] R[100]mm/sec CNT100 TB   .50sec,CALL END_PUD;
   1:  DO[117:Laser Start]=OFF;
   1:  PR[92] = PR[91];
   1:  PR[92,3] = PR[92,3] + 50;
   1:J PR[92] 10% FINE;
   1:  WAIT   5.00(sec);
   1:  DO[119:Gas]=OFF;
   1:  CALL HOME_ALL;
/POS
/END
